FUNCTION_BLOCK AxisEnableCommand IMPLEMENTS ITF_Command
VAR
END_VAR

{warning 'add method implementation '}
METHOD Execute : BOOL
END_METHOD

END_FUNCTION_BLOCK

(* stored: Version 1.1.0.1, ProductVersion 3.1.4024.12
   POU AxisEnableCommand: Id {ae9910ac-db5f-4311-ac9c-6542f482a03c}, SpecialFunc None
   Method Execute: Id {a6736136-4204-4350-9dc3-76fdcacf942b} *)
